TYPE ST_SYSTEM_ProductionLine :
STRUCT
	sPCM			: STRING(4);
	sMENo			: STRING(5);
	nTopologyID	: INT;
END_STRUCT
END_TYPE

(* stored: Version 1.1.0.1, ProductVersion 3.1.4024.15
   DUT ST_SYSTEM_ProductionLine: Id {2a7531ce-5163-45a0-b470-9f3d82161e64} *)
